// TwinCAT 3 PLC project Buttons
// ProgramVersion: 3.1.4024.0
// libraries:
//   Tc2_Standard, * (Beckhoff Automation GmbH)
//   Tc2_System, * (Beckhoff Automation GmbH)
//   Tc3_Module, * (Beckhoff Automation GmbH)
//   VisuDialogs, * (System)
// project tree:
//   / GlobalTextList.TcGTLO, PlcTask.TcTTO, Visualization Manager.TcVMO (not stored)
//   POUs/ FB_OnAndOffButtons.TcPOU, FB_PressedButton.TcPOU, FB_TimedButton.TcPOU, FB_ToggleButton.TcPOU, MAIN.TcPOU
//   VISUs/ Visualization.TcVIS
// real-time tasks:
//   TASK PlcTask: cycle T#10ms, priority 20, ADS port 350

CONFIGURATION Buttons
    RESOURCE PLC ON TwinCAT3
        TASK PlcTask(INTERVAL := T#10ms, PRIORITY := 20);
        PROGRAM MAIN WITH PlcTask : MAIN;
    END_RESOURCE
END_CONFIGURATION

// ---- POUs/MAIN.TcPOU
PROGRAM MAIN
VAR
	// Instances of appropriate FBs
	fbPressedButton : FB_PressedButton;
	fbOnAndOffButtons : FB_OnAndOffButtons;
	fbToggleButton : FB_ToggleButton;
	fbTimedButton : FB_TimedButton;

	// To know whether we've pressed certain buttons
	bIsButtonPressed : BOOL;
	bIsButtonOn : BOOL;
	bIsButtonOff : BOOL;
	bIsToggleButtonOn : BOOL;
	bIsTimeButtonPressed : BOOL;
END_VAR
VAR CONSTANT
	T_MAX_TIME : TIME;	// Max time for the timed button
END_VAR

// Calling of FBs with info we're getting from the buttons (whether they're being pressed or not)
fbPressedButton(bIsButtonPressed := bIsButtonPressed);

fbOnAndOffButtons(bIsButtonOn := bIsButtonOn, bIsButtonOff := bIsButtonOff);

fbToggleButton(bIsToggleButtonOn := bIsToggleButtonOn);

fbTimedButton(bIsTimeButtonPressed := bIsTimeButtonPressed, tMaxTime := T_MAX_TIME);

END_PROGRAM

// ---- POUs/FB_PressedButton.TcPOU
FUNCTION_BLOCK FB_PressedButton
VAR_INPUT
	bIsButtonPressed : BOOL;
END_VAR
VAR_OUTPUT
	bLightOfPressedButton : BOOL;
END_VAR
VAR
END_VAR

// As long as the button is pressed the light is on, when it's not pressed, light turns off
IF bIsButtonPressed THEN
	bLightOfPressedButton := TRUE;
ELSE
	bLightOfPressedButton := FALSE;
END_IF

END_FUNCTION_BLOCK

// ---- POUs/FB_OnAndOffButtons.TcPOU
FUNCTION_BLOCK FB_OnAndOffButtons
VAR_INPUT
	bIsButtonOn : BOOL;
	bIsButtonOff : BOOL;
END_VAR
VAR_OUTPUT
	bLightOfOnAndOffButton : BOOL;
END_VAR
VAR
	fbOn_RTRIG : R_TRIG;
	fbOff_RTRIG : R_TRIG;
END_VAR

// One button turns the light on, the other turns it off
IF bIsButtonOn THEN
	bLightOfOnAndOffButton := TRUE;
	bIsButtonOff := FALSE;
END_IF

IF bIsButtonOff THEN
	bLightOfOnAndOffButton := FALSE;
	bIsButtonOn := FALSE;
END_IF

// Solution using triggers:
//fbOn_RTRIG(clk := bIsButtonOn);
//IF fbOn_RTRIG.Q THEN
//	bLightOfOnAndOffButton := TRUE;
//	fbOn_RTRIG(clk := FALSE);
//END_IF

//fbOff_RTRIG(clk := bIsButtonOff);
//IF fbOff_RTRIG.Q THEN
//	bLightOfOnAndOffButton := FALSE;
//	fbOff_RTRIG(clk := FALSE);
//END_IF

END_FUNCTION_BLOCK

// ---- POUs/FB_ToggleButton.TcPOU
FUNCTION_BLOCK FB_ToggleButton
VAR_INPUT
	bIsToggleButtonOn : BOOL;
END_VAR
VAR_OUTPUT
	bLightOfToggleButton : BOOL;
END_VAR
VAR
	fbToggle_RTRIG : R_TRIG;
END_VAR

// When a button is clicked, turn light on if it was off, or turn light off if it was on
fbToggle_RTRIG(clk := bIsToggleButtonOn);
IF fbToggle_RTRIG.Q THEN
	bLightOfToggleButton := NOT bLightOfToggleButton;
END_IF

END_FUNCTION_BLOCK

// ---- POUs/FB_TimedButton.TcPOU
FUNCTION_BLOCK FB_TimedButton
VAR_INPUT
	bIsTimeButtonPressed : BOOL;
	tMaxTime : TIME;	// Maximum time to hold the button before swithing lights
END_VAR
VAR_OUTPUT
	bLightOfTimedButton : BOOL;
	bLightOfOtherButton : BOOL;
END_VAR
VAR
	fbTimerForTimedButton : TON;	// For timing the button press
	tTimePressed : DWORD;
	
	sMaxTime : DWORD := 3000;
END_VAR

IF bIsTimeButtonPressed  THEN	// Check if the time button is pressed
	tMaxTime := DWORD_TO_TIME(sMaxTime);
	fbTimerForTimedButton(IN := TRUE, PT := tMaxTime);	// Start the timer
	tTimePressed := TIME_TO_DWORD(fbTimerForTimedButton.ET);
	// If timer hasn't reached max time, turn on first light, ensure second light is off
	IF NOT fbTimerForTimedButton.Q THEN
		bLightOfTimedButton := TRUE;
		bLightOfOtherButton := FALSE;
	// If timer has reached max time, turn off first light, turn on second light
	ELSE
		bLightOfTimedButton := FALSE;
		bLightOfOtherButton := TRUE;
	END_IF
ELSE	// Button is not pressed
	fbTimerForTimedButton(IN := FALSE);	// Reset the timer
	// Both lights should be off
	bLightOfTimedButton := FALSE;
	bLightOfOtherButton := FALSE;
END_IF

END_FUNCTION_BLOCK

// ---- GlobalTextList.TcGTLO
TEXTLIST GlobalTextList
  602 = 'Bulb 1'
  239 = 'Bulb 2'
  308 = 'Bulb 3'
  550 = 'Bulb 4'
  952 = 'Button 1'
  404 = 'Change max time (in ms) here'
  331 = 'Change max time here'
  408 = 'Change max time here (in miliseconds)'
  139 = 'Change max time here (in ms)'
  750 = 'First light has been on for'
  73 = 'First light has been on for %s'
  989 = 'First light has been on for %s ms'
  804 = 'First light has been on for %t'
  471 = 'Off Button'
  470 = 'Off button'
  304 = 'On Button'
  175 = 'On button'
  389 = 'Pressed Button'
  45 = 'Timed Bulb'
  388 = 'Timed Button'
  618 = 'Toggle Button'
  234 = "You've been pressing for %s"
END_TEXTLIST

// ---- VISUs/Visualization.TcVIS
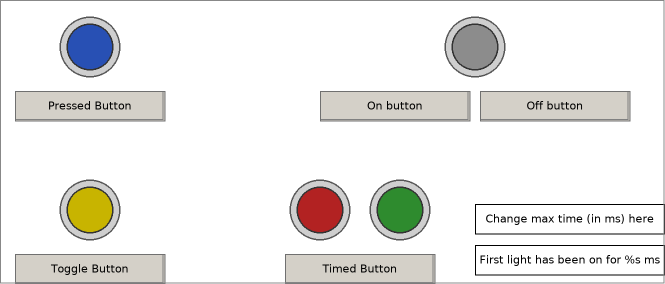
VISUALIZATION Visualization  // 665x284
    Button (15,91 150x30), "Pressed Button"
        tap MAIN.bIsButtonPressed
    Button (15,254 150x30), "Toggle Button", pressed state: main.bIsToggleButtonOn
        tap MAIN.bIsToggleButtonOn
    Button (285,254 150x30), "Timed Button"
        tap main.bIsTimeButtonPressed
    Lamp1 (55,12 70x70), variable: MAIN.fbPressedButton.bLightOfPressedButton, style: Lamp-Lamp1-Blue
    Lamp1 (440,12 70x70), variable: MAIN.fbOnAndOffButtons.bLightOfOnAndOffButton, style: Lamp-Lamp1-Gray
    Lamp1 (55,175 70x70), variable: MAIN.fbToggleButton.bLightOfToggleButton, style: Lamp-Lamp1-Yellow
    Lamp1 (285,175 70x70), variable: MAIN.fbTimedButton.bLightOfTimedButton, style: Lamp-Lamp1-Red
    Lamp1 (365,175 70x70), variable: MAIN.fbTimedButton.bLightOfOtherButton, style: Lamp-Lamp1-Green
    Rectangle (475,245 190x30), "First light has been on for %s ms", text variable: MAIN.fbTimedButton.tTimePressed
    Rectangle (475,204 190x30), "Change max time (in ms) here"
        OnMouseClick: write MAIN.fbTimedButton.sMaxTime via Default
    Button (320,91 150x30), "On button"
        tap MAIN.bIsButtonOn
    Button (480,91 150x30), "Off button"
        tap MAIN.bIsButtonOff
END_VISUALIZATION
